FUNCTION AssertNearlyEquals : BOOL
VAR_INPUT
    Source   : T_MaxString;
    Expected : LREAL;
    Actual   : LREAL;
	Delta : LREAL;
    Message  : T_MaxString;
END_VAR
VAR_OUTPUT
    Failed : BOOL;
END_VAR

IF ABS(Expected - Actual) > Delta THEN
    F_LogResult(Source, FormatStringEx1('Assertion Failed - %s', Message));
    Failed := TRUE;
    RETURN;
END_IF

AssertNearlyEquals := TRUE;

END_FUNCTION

(* stored: Version 1.1.0.1, ProductVersion 3.1.4024.11
   POU AssertNearlyEquals: Id {d9a01481-b59d-41f5-985c-6df650c93c6a}, SpecialFunc None *)
